FUNCTION_BLOCK watertank
  (* Standard: 61499-2 *)
  (* Version 0.1, 2017-00-25, hpea485, UOA *)
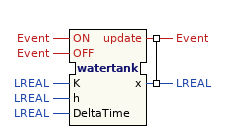
  EVENT_INPUT
    ON;
    OFF;
  END_EVENT
  EVENT_OUTPUT
    update WITH x;
  END_EVENT
  VAR_INPUT
    K : LREAL := 0.075;
    h : LREAL := 150;
    DeltaTime : LREAL := 0.01;
  END_VAR
  VAR_OUTPUT
    x : LREAL;
  END_VAR
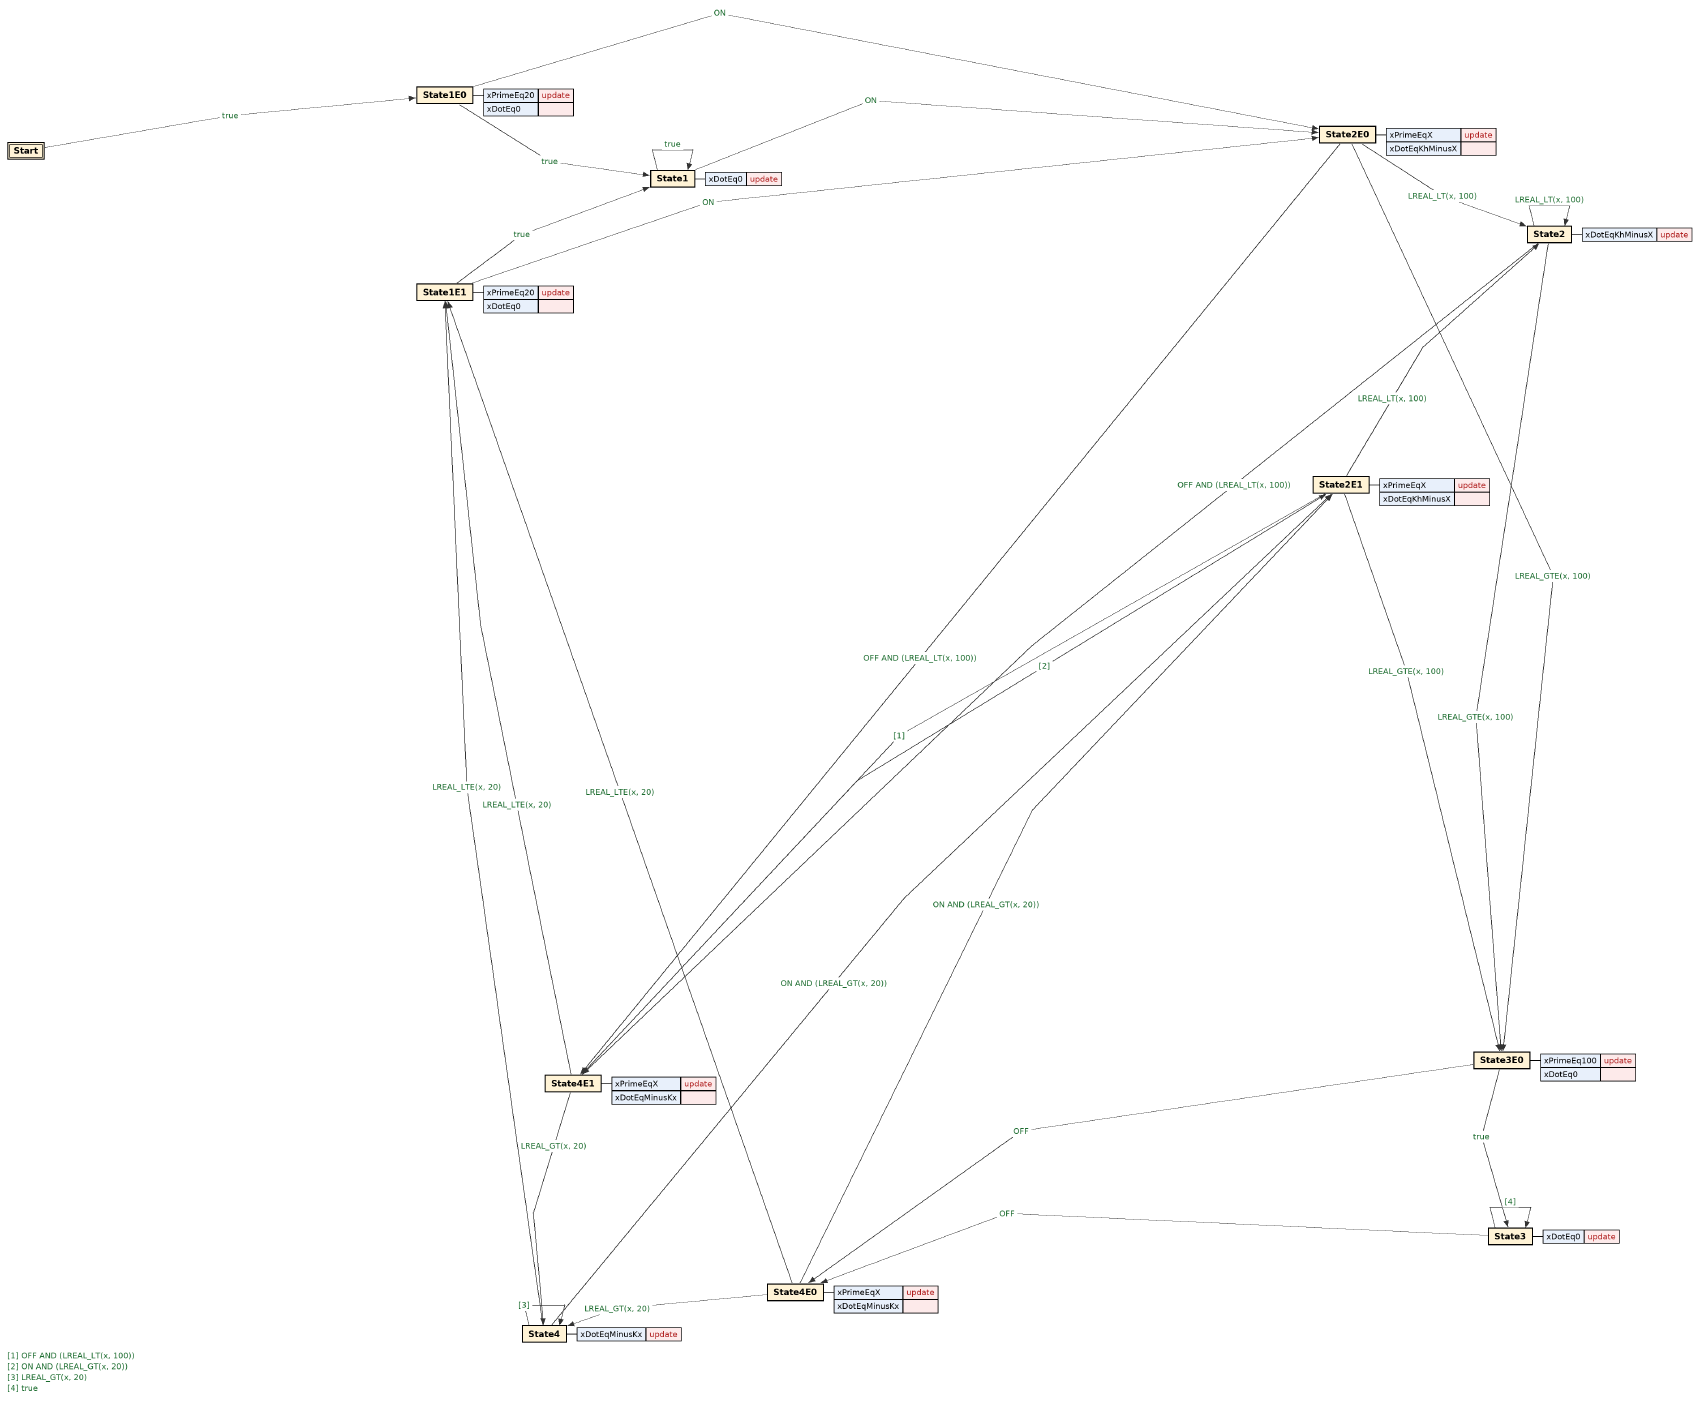
  EC_STATES
    Start;
    State1E0 : xPrimeEq20 -> update, xDotEq0;
    State1 : xDotEq0 -> update;
    State2E0 : xPrimeEqX -> update, xDotEqKhMinusX;
    State2 : xDotEqKhMinusX -> update;
    State3E0 : xPrimeEq100 -> update, xDotEq0;
    State3 : xDotEq0 -> update;
    State4E0 : xPrimeEqX -> update, xDotEqMinusKx;
    State4 : xDotEqMinusKx -> update;
    State2E1 : xPrimeEqX -> update, xDotEqKhMinusX;
    State4E1 : xPrimeEqX -> update, xDotEqMinusKx;
    State1E1 : xPrimeEq20 -> update, xDotEq0;
  END_STATES
  EC_TRANSITIONS
    Start TO State1E0 := true;
    State1E0 TO State2E0 := ON;
    State1E0 TO State1 := true;
    State1 TO State2E0 := ON;
    State1 TO State1 := true;
    State2E0 TO State3E0 := LREAL_GTE(x, 100);
    State2E0 TO State4E1 := OFF AND (LREAL_LT(x, 100));
    State2E0 TO State2 := LREAL_LT(x, 100);
    State2 TO State3E0 := LREAL_GTE(x, 100);
    State2 TO State4E1 := OFF AND (LREAL_LT(x, 100));
    State2 TO State2 := LREAL_LT(x, 100);
    State3E0 TO State4E0 := OFF;
    State3E0 TO State3 := true;
    State3 TO State4E0 := OFF;
    State3 TO State3 := true;
    State4E0 TO State1E1 := LREAL_LTE(x, 20);
    State4E0 TO State2E1 := ON AND (LREAL_GT(x, 20));
    State4E0 TO State4 := LREAL_GT(x, 20);
    State4 TO State1E1 := LREAL_LTE(x, 20);
    State4 TO State2E1 := ON AND (LREAL_GT(x, 20));
    State4 TO State4 := LREAL_GT(x, 20);
    State2E1 TO State3E0 := LREAL_GTE(x, 100);
    State2E1 TO State4E1 := OFF AND (LREAL_LT(x, 100));
    State2E1 TO State2 := LREAL_LT(x, 100);
    State4E1 TO State1E1 := LREAL_LTE(x, 20);
    State4E1 TO State2E1 := ON AND (LREAL_GT(x, 20));
    State4E1 TO State4 := LREAL_GT(x, 20);
    State1E1 TO State2E0 := ON;
    State1E1 TO State1 := true;
  END_TRANSITIONS
  ALGORITHM xPrimeEq20 IN C: (* ODE_init *)
x_prime = 20;
  END_ALGORITHM
  ALGORITHM xPrimeEqX IN C: (* ODE_init *)
x_prime = x;
  END_ALGORITHM
  ALGORITHM xDotEq0 IN C: (* ODE *)
x_dot = 0;
  END_ALGORITHM
  ALGORITHM xDotEqMinusKx IN C: (* ODE *)
x_dot = -K * x;x_trigger = 20;
  END_ALGORITHM
  ALGORITHM xDotEqKhMinusX IN C: (* ODE *)
x_dot = K * (h - x);
x_trigger = 100;
  END_ALGORITHM
  ALGORITHM xPrimeEq100 IN C: (* ODE_init *)
x_prime = 100;
  END_ALGORITHM
END_FUNCTION_BLOCK
